{attribute 'GeneratedUsingTerminal: ELX3181-0000-0016'}
{attribute addProperty BoxType "ELX3181-0000-0016"}
{attribute addProperty Id "Ch_1Ch_1_A1FAE75910WcStateAT %I*WcState_9091E0EB2InfoDataAT %I*InfoData_41C547A32"}
{attribute addProperty CRC "3567561197"}
{attribute addProperty Size "14"}
TYPE ELX3181_D4A4A9ED EXTENDS EtcSlaveTerminalBase_947E5A46 :
STRUCT
	{attribute addProperty Name "Ch_1"}
	Ch_1 : Ch_1_A1FAE759;
	{attribute addProperty Name "WcState"}
	WcState : WcState_9091E0EB;
	{attribute addProperty Name "InfoData"}
	InfoData : InfoData_41C547A3;
END_STRUCT
END_TYPE

(* stored: Version 1.2.0.0, ProductVersion 3.1.4024.9
   DUT ELX3181_D4A4A9ED: Id {c7ce097a-5775-4bdb-a18e-b0dbbb27ebe4} *)
